(* IEC 61131-3 sources: netRob/Hardwareadapter/robot/functions, 4 files *)

(* ---- MoveToPos.ST ---- *)
(*@PROPERTIES_EX@
TYPE: POU
LOCALE: 0
IEC_LANGUAGE: ST
PLC_TYPE: independent
PROC_TYPE: independent
*)
(*@KEY@:DESCRIPTION*)

(*@KEY@:END_DESCRIPTION*)
FUNCTION_BLOCK MoveToPos
VAR_INPUT
	x: LREAL;
	y: LREAL;
	z: LREAL;
	u: LREAL;
END_VAR
VAR_IN_OUT
	completed: BOOL;
END_VAR
VAR
	move_x: MC_MoveAbsolute;
	move_y: MC_MoveAbsolute;
	move_z: MC_MoveAbsolute;
	move_u: MC_MoveAbsolute;
END_VAR

(*@KEY@: WORKSHEET
NAME: MoveToPos
IEC_LANGUAGE: ST
*)
move_x(Axis:=CMMT_AS_X,Execute:=TRUE,Position:=x,Velocity:=100,Acceleration:=1000,Deceleration:=1000,Jerk:=10000);
move_y(Axis:=CMMT_AS_Y,Execute:=TRUE,Position:=y,Velocity:=100,Acceleration:=1000,Deceleration:=1000,Jerk:=10000);
move_z(Axis:=CMMT_AS_Z,Execute:=TRUE,Position:=z,Velocity:=50,Acceleration:=1000,Deceleration:=1000,Jerk:=10000);
move_u(Axis:=CMMT_ST_U,Execute:=TRUE,Position:=u,Velocity:=100,Acceleration:=1000,Deceleration:=1000,Jerk:=10000);

IF move_x.Done = TRUE AND move_y.Done = TRUE AND move_z.Done = TRUE AND move_u.Done = TRUE THEN
	move_x(Axis:=CMMT_AS_X,Execute:=FALSE);
	move_y(Axis:=CMMT_AS_Y,Execute:=FALSE);
	move_z(Axis:=CMMT_AS_Z,Execute:=FALSE);
	move_u(Axis:=CMMT_ST_U,Execute:=FALSE);
	completed := TRUE;
END_IF
(*@KEY@: END_WORKSHEET *)
END_FUNCTION_BLOCK

(* ---- PowerUp.ST ---- *)
(*@PROPERTIES_EX@
TYPE: POU
LOCALE: 0
IEC_LANGUAGE: ST
PLC_TYPE: independent
PROC_TYPE: independent
*)
(*@KEY@:DESCRIPTION*)

(*@KEY@:END_DESCRIPTION*)
FUNCTION_BLOCK PowerUp
VAR_IN_OUT
	completed: BOOL; (* Indicates if all axes have completed the startup phase.*)
END_VAR
VAR
	power_x: MC_Power;
	power_y: MC_Power;
	power_z: MC_Power;
	power_u: MC_Power;
END_VAR

(*@KEY@: WORKSHEET
NAME: PowerUp
IEC_LANGUAGE: ST
*)
power_x(Axis:=CMMT_AS_X,Enable:=TRUE,bRegulatorOn:=TRUE,bdriveStart:=TRUE);
power_y(Axis:=CMMT_AS_Y,Enable:=TRUE,bRegulatorOn:=TRUE,bdriveStart:=TRUE);
power_z(Axis:=CMMT_AS_Z,Enable:=TRUE,bRegulatorOn:=TRUE,bdriveStart:=TRUE);
power_u(Axis:=CMMT_ST_U,Enable:=TRUE,bRegulatorOn:=TRUE,bdriveStart:=TRUE);

IF power_x.Status = TRUE AND power_y.Status = TRUE AND power_z.Status = TRUE AND power_u.Status = TRUE THEN
	completed := TRUE;
END_IF
(*@KEY@: END_WORKSHEET *)
END_FUNCTION_BLOCK

(* ---- ResetAxisErrors.ST ---- *)
(*@PROPERTIES_EX@
TYPE: POU
LOCALE: 0
IEC_LANGUAGE: ST
PLC_TYPE: independent
PROC_TYPE: independent
*)
(*@KEY@:DESCRIPTION*)

(*@KEY@:END_DESCRIPTION*)
FUNCTION_BLOCK ResetAxisErrors
VAR_INPUT
END_VAR
VAR_OUTPUT
	completed: BOOL; (* indicates whether error resetting has been completed *)
END_VAR
VAR
	reset_x: MC_Reset;
	reset_y: MC_Reset;
	reset_z: MC_Reset;
	reset_u: MC_Reset;
END_VAR

(*@KEY@: WORKSHEET
NAME: ResetAxisErrors
IEC_LANGUAGE: ST
*)
reset_x(Axis:=CMMT_AS_X,Execute:=TRUE);
reset_y(Axis:=CMMT_AS_Y,Execute:=TRUE);
reset_z(Axis:=CMMT_AS_Z,Execute:=TRUE);
reset_u(Axis:=CMMT_ST_U,Execute:=TRUE);
IF reset_x.Done = TRUE AND reset_y.Done = TRUE AND reset_z.Done = TRUE AND reset_u.Done = TRUE THEN
	reset_x(Axis:=CMMT_AS_X,Execute:=FALSE);
	reset_y(Axis:=CMMT_AS_Y,Execute:=FALSE);
	reset_z(Axis:=CMMT_AS_Z,Execute:=FALSE);
	reset_u(Axis:=CMMT_ST_U,Execute:=FALSE);
	completed := TRUE;
END_IF
(*@KEY@: END_WORKSHEET *)
END_FUNCTION_BLOCK

(* ---- StopMovement.ST ---- *)
(*@PROPERTIES_EX@
TYPE: POU
LOCALE: 0
IEC_LANGUAGE: ST
PLC_TYPE: independent
PROC_TYPE: independent
*)
(*@KEY@:DESCRIPTION*)

(*@KEY@:END_DESCRIPTION*)
FUNCTION_BLOCK StopMovement
VAR_INPUT
END_VAR
VAR_IN_OUT
	completed: BOOL;
END_VAR
VAR
	stop_x: MC_Stop;
	stop_y: MC_Stop;
	stop_z: MC_Stop;
	stop_u: MC_Stop;
END_VAR

(*@KEY@: WORKSHEET
NAME: StopMovement
IEC_LANGUAGE: ST
*)
stop_x(Axis:=CMMT_AS_X,Execute:=TRUE,Deceleration:=1000,Jerk:=100000);
stop_y(Axis:=CMMT_AS_Y,Execute:=TRUE,Deceleration:=1000,Jerk:=100000);
stop_z(Axis:=CMMT_AS_Z,Execute:=TRUE,Deceleration:=1000,Jerk:=100000);
stop_u(Axis:=CMMT_ST_U,Execute:=TRUE,Deceleration:=1000,Jerk:=100000);

IF stop_x.Done = TRUE AND stop_y.Done = TRUE AND stop_z.Done = TRUE AND stop_u.Done = TRUE THEN
	stop_x(Axis:=CMMT_AS_X,Execute:=FALSE);
	stop_y(Axis:=CMMT_AS_Y,Execute:=FALSE);
	stop_z(Axis:=CMMT_AS_Z,Execute:=FALSE);
	stop_u(Axis:=CMMT_ST_U,Execute:=FALSE);
	completed := TRUE;
END_IF
(*@KEY@: END_WORKSHEET *)
END_FUNCTION_BLOCK
